// TIA Portal V17 export
// export: Created 2024-09-02T12:50:15.0745708Z, ExportSetting WithDefaults, DisplayName Totally Integrated Automation Portal, DisplayVersion V17, DisplayName TIA Portal Openness, DisplayVersion V17, DisplayName TIA Portal Version Control Interface, DisplayVersion V17, DisplayName STEP 7 Professional, DisplayVersion V17, DisplayName STEP 7 Safety, DisplayVersion V17, DisplayName WinCC Professional, DisplayVersion V17
FUNCTION "AnwFC_ZP_OperatingModes_OP70" : Void   // FC61, LAD
TITLE = FC Operating modes / FC Betriebsarten
{ S7_Optimized_Access := 'TRUE' }
AUTHOR : OlegFuehrus
FAMILY : BA
NAME : BA
VERSION : 0.0
// stored: AutoNumber true, IsIECCheckEnabled false, SetENOAutomatically false, UDAEnableTagReadback false
   VAR_TEMP
      t_e_stop_ok : Bool;
      Dummy : Bool;
   END_VAR
   VAR_TEMP   // added for the SCL form of the ladder/FBD networks
      _w1 : Bool;
      _w2 : Bool;
      _w3 : Bool;
      _w4 : Bool;
      _w5 : Bool;
      _w6 : Bool;
   END_VAR
BEGIN

REGION Network 1: Station lighting On / Stationbeleuchtung Ein
END_REGION

REGION Network 2: Maschine Off (+S-KFK0) / Maschine Aus (+S-KFK0)
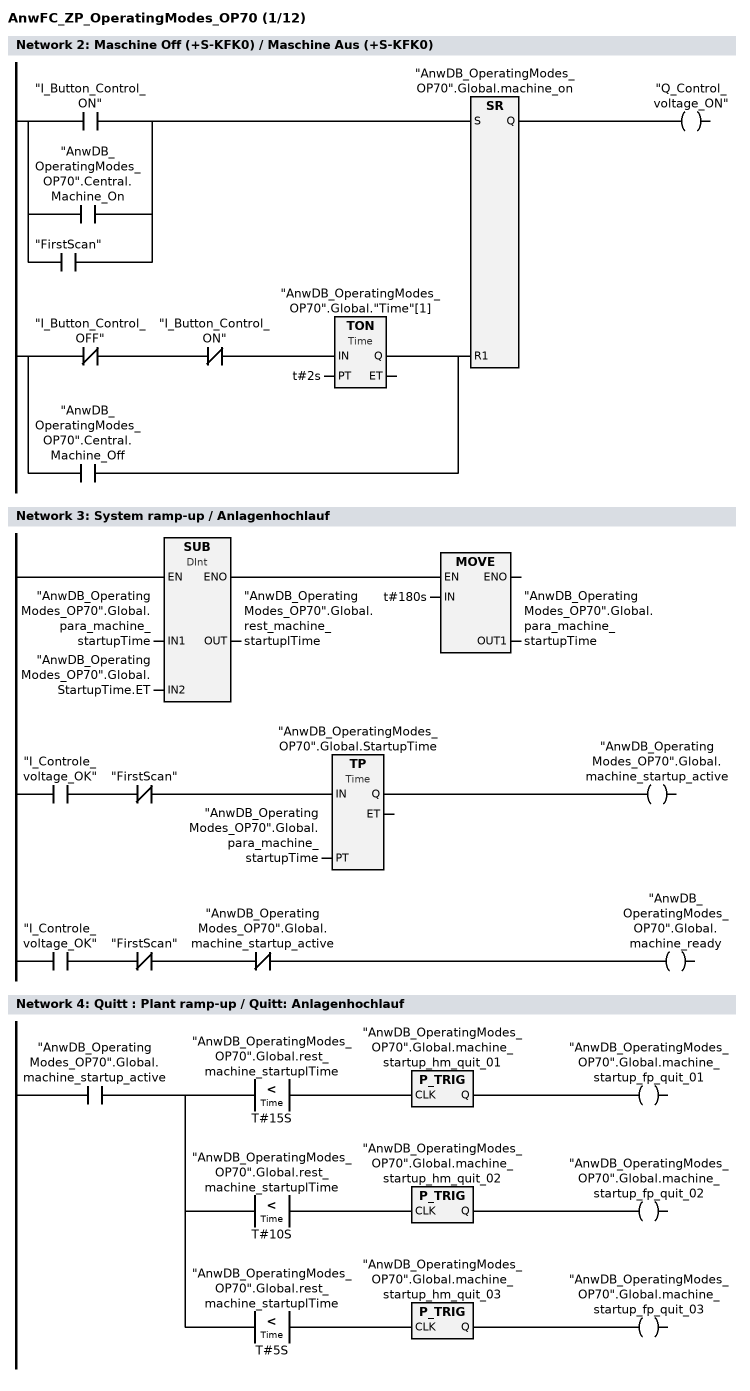
   RUNG wire#powerrail
      Contact( "I_Button_Control_ON" )
      wire#w1
      S_SR(operand := "AnwDB_OperatingModes_OP70".Global.machine_on, r1 := wire#w2)
      Coil( "Q_Control_voltage_ON" )
   END_RUNG
   RUNG wire#powerrail
      Contact( "AnwDB_OperatingModes_OP70".Central.Machine_On )
   END_RUNG wire#w1
   RUNG wire#powerrail
      Contact( "FirstScan" )
   END_RUNG wire#w1
   RUNG wire#powerrail
      I_Contact( "I_Button_Control_OFF" )
      I_Contact( "I_Button_Control_ON" )
      { S7_Templates := "time_type := Time" } "AnwDB_OperatingModes_OP70".Global."Time"[1].TON(pt := t#2s, et =>)
   END_RUNG wire#w2
   RUNG wire#powerrail
      Contact( "AnwDB_OperatingModes_OP70".Central.Machine_Off )
   END_RUNG wire#w2
   // the same network as SCL:
   "AnwDB_OperatingModes_OP70".Global."Time"[1].TON(IN := NOT "I_Button_Control_OFF" AND NOT "I_Button_Control_ON",
                           PT := t#2s);
   IF "I_Button_Control_ON" OR "AnwDB_OperatingModes_OP70".Central.Machine_On OR "FirstScan" THEN
       "AnwDB_OperatingModes_OP70".Global.machine_on := TRUE;   // SR flip-flop
   END_IF;
   IF "AnwDB_OperatingModes_OP70".Global."Time"[1].Q OR "AnwDB_OperatingModes_OP70".Central.Machine_Off THEN
       "AnwDB_OperatingModes_OP70".Global.machine_on := FALSE;
   END_IF;
   "Q_Control_voltage_ON" := "AnwDB_OperatingModes_OP70".Global.machine_on;
END_REGION

REGION Network 3: System ramp-up / Anlagenhochlauf
   RUNG wire#powerrail
      { S7_Templates := "SrcType := DInt" } Sub(in1 := "AnwDB_OperatingModes_OP70".Global.para_machine_startupTime, in2 := "AnwDB_OperatingModes_OP70".Global.StartupTime.ET, out => "AnwDB_OperatingModes_OP70".Global.rest_machine_startuplTime)
      Move(in := t#180s, out1 => "AnwDB_OperatingModes_OP70".Global.para_machine_startupTime)
   END_RUNG
   RUNG wire#powerrail
      Contact( "I_Controle_voltage_OK" )
      I_Contact( "FirstScan" )
      { S7_Templates := "time_type := Time" } "AnwDB_OperatingModes_OP70".Global.StartupTime.TP(pt := "AnwDB_OperatingModes_OP70".Global.para_machine_startupTime, et =>)
      Coil( "AnwDB_OperatingModes_OP70".Global.machine_startup_active )
   END_RUNG
   RUNG wire#powerrail
      Contact( "I_Controle_voltage_OK" )
      I_Contact( "FirstScan" )
      I_Contact( "AnwDB_OperatingModes_OP70".Global.machine_startup_active )
      Coil( "AnwDB_OperatingModes_OP70".Global.machine_ready )
   END_RUNG
   // the same network as SCL:
   "AnwDB_OperatingModes_OP70".Global.rest_machine_startuplTime := "AnwDB_OperatingModes_OP70".Global.para_machine_startupTime - "AnwDB_OperatingModes_OP70".Global.StartupTime.ET;
   "AnwDB_OperatingModes_OP70".Global.para_machine_startupTime := t#180s;
   "AnwDB_OperatingModes_OP70".Global.StartupTime.TP(IN := "I_Controle_voltage_OK" AND NOT "FirstScan",
                           PT := "AnwDB_OperatingModes_OP70".Global.para_machine_startupTime);
   "AnwDB_OperatingModes_OP70".Global.machine_startup_active := "AnwDB_OperatingModes_OP70".Global.StartupTime.Q;
   "AnwDB_OperatingModes_OP70".Global.machine_ready := "I_Controle_voltage_OK" AND NOT "FirstScan" AND NOT "AnwDB_OperatingModes_OP70".Global.machine_startup_active;
END_REGION

REGION Network 4: Quitt : Plant ramp-up / Quitt: Anlagenhochlauf
   RUNG wire#powerrail
      Contact( "AnwDB_OperatingModes_OP70".Global.machine_startup_active )
      wire#w1
      { S7_Templates := "SrcType := Time" } LT_Contact(in1 := "AnwDB_OperatingModes_OP70".Global.rest_machine_startuplTime, in2 := T#15S)
      P_Trig( "AnwDB_OperatingModes_OP70".Global.machine_startup_hm_quit_01 )
      Coil( "AnwDB_OperatingModes_OP70".Global.machine_startup_fp_quit_01 )
   END_RUNG
   RUNG wire#w1
      { S7_Templates := "SrcType := Time" } LT_Contact(in1 := "AnwDB_OperatingModes_OP70".Global.rest_machine_startuplTime, in2 := T#10S)
      P_Trig( "AnwDB_OperatingModes_OP70".Global.machine_startup_hm_quit_02 )
      Coil( "AnwDB_OperatingModes_OP70".Global.machine_startup_fp_quit_02 )
   END_RUNG
   RUNG wire#w1
      { S7_Templates := "SrcType := Time" } LT_Contact(in1 := "AnwDB_OperatingModes_OP70".Global.rest_machine_startuplTime, in2 := T#5S)
      P_Trig( "AnwDB_OperatingModes_OP70".Global.machine_startup_hm_quit_03 )
      Coil( "AnwDB_OperatingModes_OP70".Global.machine_startup_fp_quit_03 )
   END_RUNG
   // the same network as SCL:
   #_w1 := "AnwDB_OperatingModes_OP70".Global.machine_startup_active AND ("AnwDB_OperatingModes_OP70".Global.rest_machine_startuplTime < T#15S);
   #_w2 := #_w1 AND NOT "AnwDB_OperatingModes_OP70".Global.machine_startup_hm_quit_01;   // rising edge
   "AnwDB_OperatingModes_OP70".Global.machine_startup_hm_quit_01 := #_w1;
   "AnwDB_OperatingModes_OP70".Global.machine_startup_fp_quit_01 := #_w2;
   #_w3 := "AnwDB_OperatingModes_OP70".Global.machine_startup_active AND ("AnwDB_OperatingModes_OP70".Global.rest_machine_startuplTime < T#10S);
   #_w4 := #_w3 AND NOT "AnwDB_OperatingModes_OP70".Global.machine_startup_hm_quit_02;   // rising edge
   "AnwDB_OperatingModes_OP70".Global.machine_startup_hm_quit_02 := #_w3;
   "AnwDB_OperatingModes_OP70".Global.machine_startup_fp_quit_02 := #_w4;
   #_w5 := "AnwDB_OperatingModes_OP70".Global.machine_startup_active AND ("AnwDB_OperatingModes_OP70".Global.rest_machine_startuplTime < T#5S);
   #_w6 := #_w5 AND NOT "AnwDB_OperatingModes_OP70".Global.machine_startup_hm_quit_03;   // rising edge
   "AnwDB_OperatingModes_OP70".Global.machine_startup_hm_quit_03 := #_w5;
   "AnwDB_OperatingModes_OP70".Global.machine_startup_fp_quit_03 := #_w6;
END_REGION

REGION Network 5: Starting conditions Ready / Startvoraussetzungen Bereit
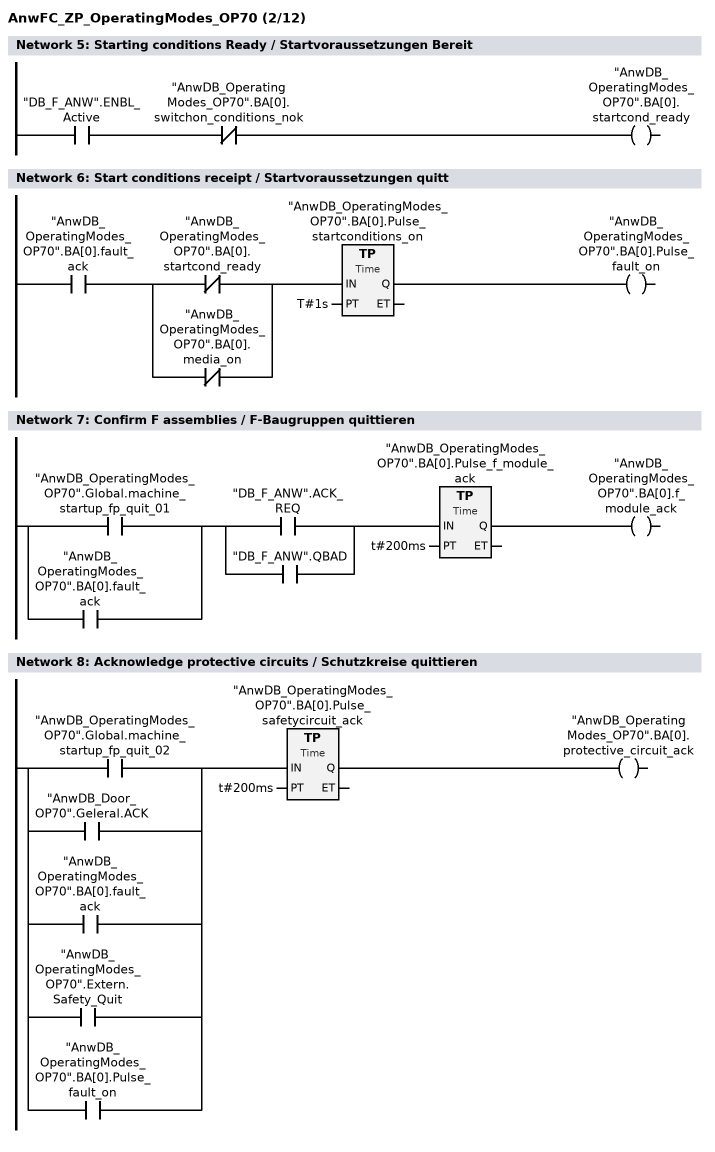
   RUNG wire#powerrail
      Contact( "DB_F_ANW".ENBL_Active )
      I_Contact( "AnwDB_OperatingModes_OP70".BA[0].switchon_conditions_nok )
      Coil( "AnwDB_OperatingModes_OP70".BA[0].startcond_ready )
   END_RUNG
   // the same network as SCL:
   "AnwDB_OperatingModes_OP70".BA[0].startcond_ready := "DB_F_ANW".ENBL_Active AND NOT "AnwDB_OperatingModes_OP70".BA[0].switchon_conditions_nok;
END_REGION

REGION Network 6: Start conditions receipt / Startvoraussetzungen quitt
   RUNG wire#powerrail
      Contact( "AnwDB_OperatingModes_OP70".BA[0].fault_ack )
      wire#w1
      I_Contact( "AnwDB_OperatingModes_OP70".BA[0].startcond_ready )
      wire#w2
      { S7_Templates := "time_type := Time" } "AnwDB_OperatingModes_OP70".BA[0].Pulse_startconditions_on.TP(pt := T#1s, et =>)
      Coil( "AnwDB_OperatingModes_OP70".BA[0].Pulse_fault_on )
   END_RUNG
   RUNG wire#w1
      I_Contact( "AnwDB_OperatingModes_OP70".BA[0].media_on )
   END_RUNG wire#w2
   // the same network as SCL:
   "AnwDB_OperatingModes_OP70".BA[0].Pulse_startconditions_on.TP(IN := "AnwDB_OperatingModes_OP70".BA[0].fault_ack AND (NOT "AnwDB_OperatingModes_OP70".BA[0].startcond_ready OR NOT "AnwDB_OperatingModes_OP70".BA[0].media_on),
                           PT := T#1s);
   "AnwDB_OperatingModes_OP70".BA[0].Pulse_fault_on := "AnwDB_OperatingModes_OP70".BA[0].Pulse_startconditions_on.Q;
END_REGION

REGION Network 7: Confirm F assemblies / F-Baugruppen quittieren
   RUNG wire#powerrail
      Contact( "AnwDB_OperatingModes_OP70".Global.machine_startup_fp_quit_01 )
      wire#w1
      Contact( "DB_F_ANW".ACK_REQ )
      wire#w2
      { S7_Templates := "time_type := Time" } "AnwDB_OperatingModes_OP70".BA[0].Pulse_f_module_ack.TP(pt := t#200ms, et =>)
      Coil( "AnwDB_OperatingModes_OP70".BA[0].f_module_ack )
   END_RUNG
   RUNG wire#powerrail
      Contact( "AnwDB_OperatingModes_OP70".BA[0].fault_ack )
   END_RUNG wire#w1
   RUNG wire#w1
      Contact( "DB_F_ANW".QBAD )
   END_RUNG wire#w2
   // the same network as SCL:
   "AnwDB_OperatingModes_OP70".BA[0].Pulse_f_module_ack.TP(IN := ("AnwDB_OperatingModes_OP70".Global.machine_startup_fp_quit_01 OR "AnwDB_OperatingModes_OP70".BA[0].fault_ack) AND ("DB_F_ANW".ACK_REQ OR "DB_F_ANW".QBAD),
                           PT := t#200ms);
   "AnwDB_OperatingModes_OP70".BA[0].f_module_ack := "AnwDB_OperatingModes_OP70".BA[0].Pulse_f_module_ack.Q;
END_REGION

REGION Network 8: Acknowledge protective circuits / Schutzkreise quittieren
   RUNG wire#powerrail
      Contact( "AnwDB_OperatingModes_OP70".Global.machine_startup_fp_quit_02 )
      wire#w1
      { S7_Templates := "time_type := Time" } "AnwDB_OperatingModes_OP70".BA[0].Pulse_safetycircuit_ack.TP(pt := t#200ms, et =>)
      Coil( "AnwDB_OperatingModes_OP70".BA[0].protective_circuit_ack )
   END_RUNG
   RUNG wire#powerrail
      Contact( "AnwDB_Door_OP70".Geleral.ACK )
   END_RUNG wire#w1
   RUNG wire#powerrail
      Contact( "AnwDB_OperatingModes_OP70".BA[0].fault_ack )
   END_RUNG wire#w1
   RUNG wire#powerrail
      Contact( "AnwDB_OperatingModes_OP70".Extern.Safety_Quit )
   END_RUNG wire#w1
   RUNG wire#powerrail
      Contact( "AnwDB_OperatingModes_OP70".BA[0].Pulse_fault_on )
   END_RUNG wire#w1
   // the same network as SCL:
   "AnwDB_OperatingModes_OP70".BA[0].Pulse_safetycircuit_ack.TP(IN := "AnwDB_OperatingModes_OP70".Global.machine_startup_fp_quit_02 OR "AnwDB_Door_OP70".Geleral.ACK OR "AnwDB_OperatingModes_OP70".BA[0].fault_ack OR "AnwDB_OperatingModes_OP70".Extern.Safety_Quit OR "AnwDB_OperatingModes_OP70".BA[0].Pulse_fault_on,
                           PT := t#200ms);
   "AnwDB_OperatingModes_OP70".BA[0].protective_circuit_ack := "AnwDB_OperatingModes_OP70".BA[0].Pulse_safetycircuit_ack.Q;
END_REGION

REGION Network 9: Fault Acknowledge / Störung quitt
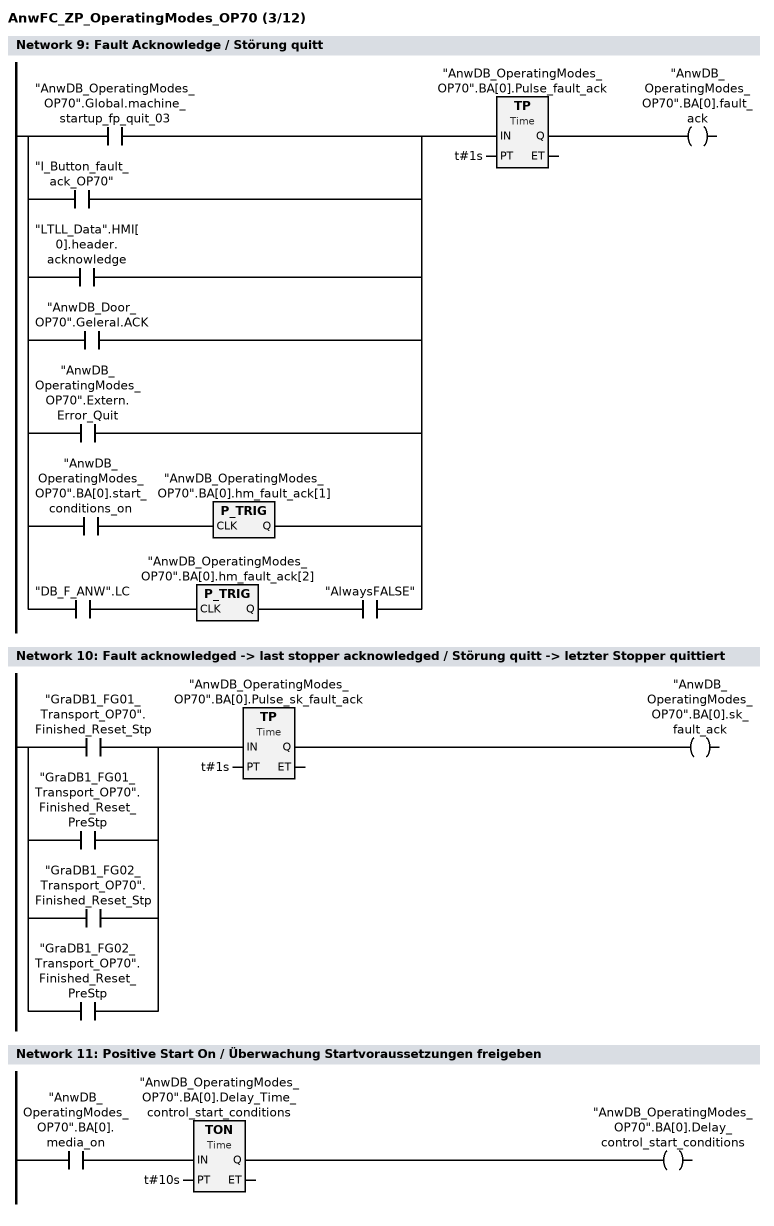
   RUNG wire#powerrail
      Contact( "AnwDB_OperatingModes_OP70".Global.machine_startup_fp_quit_03 )
      wire#w1
      { S7_Templates := "time_type := Time" } "AnwDB_OperatingModes_OP70".BA[0].Pulse_fault_ack.TP(pt := t#1s, et =>)
      Coil( "AnwDB_OperatingModes_OP70".BA[0].fault_ack )
   END_RUNG
   RUNG wire#powerrail
      Contact( "I_Button_fault_ack_OP70" )
   END_RUNG wire#w1
   RUNG wire#powerrail
      Contact( "LTLL_Data".HMI[0].header.acknowledge )
   END_RUNG wire#w1
   RUNG wire#powerrail
      Contact( "AnwDB_Door_OP70".Geleral.ACK )
   END_RUNG wire#w1
   RUNG wire#powerrail
      Contact( "AnwDB_OperatingModes_OP70".Extern.Error_Quit )
   END_RUNG wire#w1
   RUNG wire#powerrail
      Contact( "AnwDB_OperatingModes_OP70".BA[0].start_conditions_on )
      P_Trig( "AnwDB_OperatingModes_OP70".BA[0].hm_fault_ack[1] )
   END_RUNG wire#w1
   RUNG wire#powerrail
      Contact( "DB_F_ANW".LC )
      P_Trig( "AnwDB_OperatingModes_OP70".BA[0].hm_fault_ack[2] )
      Contact( "AlwaysFALSE" )
   END_RUNG wire#w1
   // the same network as SCL:
   #_w1 := "AnwDB_OperatingModes_OP70".BA[0].start_conditions_on;
   #_w2 := #_w1 AND NOT "AnwDB_OperatingModes_OP70".BA[0].hm_fault_ack[1];   // rising edge
   "AnwDB_OperatingModes_OP70".BA[0].hm_fault_ack[1] := #_w1;
   #_w3 := "DB_F_ANW".LC AND NOT "AnwDB_OperatingModes_OP70".BA[0].hm_fault_ack[2];   // rising edge
   "AnwDB_OperatingModes_OP70".BA[0].hm_fault_ack[2] := "DB_F_ANW".LC;
   "AnwDB_OperatingModes_OP70".BA[0].Pulse_fault_ack.TP(IN := "AnwDB_OperatingModes_OP70".Global.machine_startup_fp_quit_03 OR "I_Button_fault_ack_OP70" OR "LTLL_Data".HMI[0].header.acknowledge OR "AnwDB_Door_OP70".Geleral.ACK OR "AnwDB_OperatingModes_OP70".Extern.Error_Quit OR #_w2 OR (#_w3 AND "AlwaysFALSE"),
                           PT := t#1s);
   "AnwDB_OperatingModes_OP70".BA[0].fault_ack := "AnwDB_OperatingModes_OP70".BA[0].Pulse_fault_ack.Q;
END_REGION

REGION Network 10: Fault acknowledged -> last stopper acknowledged / Störung quitt -> letzter Stopper quittiert
   RUNG wire#powerrail
      Contact( "GraDB1_FG01_Transport_OP70".Finished_Reset_Stp )
      wire#w1
      { S7_Templates := "time_type := Time" } "AnwDB_OperatingModes_OP70".BA[0].Pulse_sk_fault_ack.TP(pt := t#1s, et =>)
      Coil( "AnwDB_OperatingModes_OP70".BA[0].sk_fault_ack )
   END_RUNG
   RUNG wire#powerrail
      Contact( "GraDB1_FG01_Transport_OP70".Finished_Reset_PreStp )
   END_RUNG wire#w1
   RUNG wire#powerrail
      Contact( "GraDB1_FG02_Transport_OP70".Finished_Reset_Stp )
   END_RUNG wire#w1
   RUNG wire#powerrail
      Contact( "GraDB1_FG02_Transport_OP70".Finished_Reset_PreStp )
   END_RUNG wire#w1
   // the same network as SCL:
   "AnwDB_OperatingModes_OP70".BA[0].Pulse_sk_fault_ack.TP(IN := "GraDB1_FG01_Transport_OP70".Finished_Reset_Stp OR "GraDB1_FG01_Transport_OP70".Finished_Reset_PreStp OR "GraDB1_FG02_Transport_OP70".Finished_Reset_Stp OR "GraDB1_FG02_Transport_OP70".Finished_Reset_PreStp,
                           PT := t#1s);
   "AnwDB_OperatingModes_OP70".BA[0].sk_fault_ack := "AnwDB_OperatingModes_OP70".BA[0].Pulse_sk_fault_ack.Q;
END_REGION

REGION Network 11: Positive Start On / Überwachung Startvoraussetzungen freigeben
   RUNG wire#powerrail
      Contact( "AnwDB_OperatingModes_OP70".BA[0].media_on )
      { S7_Templates := "time_type := Time" } "AnwDB_OperatingModes_OP70".BA[0].Delay_Time_control_start_conditions.TON(pt := t#10s, et =>)
      Coil( "AnwDB_OperatingModes_OP70".BA[0].Delay_control_start_conditions )
   END_RUNG
   // the same network as SCL:
   "AnwDB_OperatingModes_OP70".BA[0].Delay_Time_control_start_conditions.TON(IN := "AnwDB_OperatingModes_OP70".BA[0].media_on,
                           PT := t#10s);
   "AnwDB_OperatingModes_OP70".BA[0].Delay_control_start_conditions := "AnwDB_OperatingModes_OP70".BA[0].Delay_Time_control_start_conditions.Q;
END_REGION

REGION Network 12: Starting conditions are ON / Startvoraussetzungen sind ein
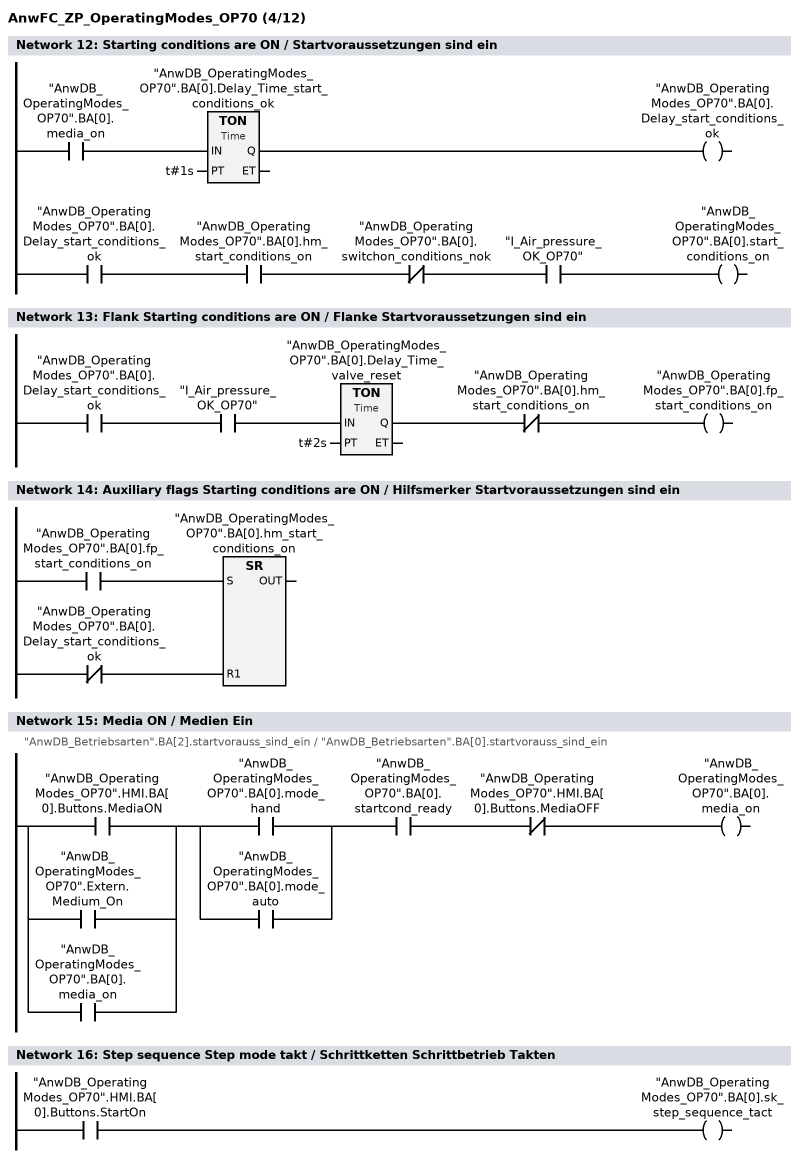
   RUNG wire#powerrail
      Contact( "AnwDB_OperatingModes_OP70".BA[0].media_on )
      { S7_Templates := "time_type := Time" } "AnwDB_OperatingModes_OP70".BA[0].Delay_Time_start_conditions_ok.TON(pt := t#1s, et =>)
      Coil( "AnwDB_OperatingModes_OP70".BA[0].Delay_start_conditions_ok )
   END_RUNG
   RUNG wire#powerrail
      Contact( "AnwDB_OperatingModes_OP70".BA[0].Delay_start_conditions_ok )
      Contact( "AnwDB_OperatingModes_OP70".BA[0].hm_start_conditions_on )
      I_Contact( "AnwDB_OperatingModes_OP70".BA[0].switchon_conditions_nok )
      Contact( "I_Air_pressure_OK_OP70" )
      Coil( "AnwDB_OperatingModes_OP70".BA[0].start_conditions_on )
   END_RUNG
   // the same network as SCL:
   "AnwDB_OperatingModes_OP70".BA[0].Delay_Time_start_conditions_ok.TON(IN := "AnwDB_OperatingModes_OP70".BA[0].media_on,
                           PT := t#1s);
   "AnwDB_OperatingModes_OP70".BA[0].Delay_start_conditions_ok := "AnwDB_OperatingModes_OP70".BA[0].Delay_Time_start_conditions_ok.Q;
   "AnwDB_OperatingModes_OP70".BA[0].start_conditions_on := "AnwDB_OperatingModes_OP70".BA[0].Delay_start_conditions_ok AND "AnwDB_OperatingModes_OP70".BA[0].hm_start_conditions_on AND NOT "AnwDB_OperatingModes_OP70".BA[0].switchon_conditions_nok AND "I_Air_pressure_OK_OP70";
END_REGION

REGION Network 13: Flank Starting conditions are ON / Flanke Startvoraussetzungen sind ein
   RUNG wire#powerrail
      Contact( "AnwDB_OperatingModes_OP70".BA[0].Delay_start_conditions_ok )
      Contact( "I_Air_pressure_OK_OP70" )
      { S7_Templates := "time_type := Time" } "AnwDB_OperatingModes_OP70".BA[0].Delay_Time_valve_reset.TON(pt := t#2s, et =>)
      I_Contact( "AnwDB_OperatingModes_OP70".BA[0].hm_start_conditions_on )
      Coil( "AnwDB_OperatingModes_OP70".BA[0].fp_start_conditions_on )
   END_RUNG
   // the same network as SCL:
   "AnwDB_OperatingModes_OP70".BA[0].Delay_Time_valve_reset.TON(IN := "AnwDB_OperatingModes_OP70".BA[0].Delay_start_conditions_ok AND "I_Air_pressure_OK_OP70",
                           PT := t#2s);
   "AnwDB_OperatingModes_OP70".BA[0].fp_start_conditions_on := "AnwDB_OperatingModes_OP70".BA[0].Delay_Time_valve_reset.Q AND NOT "AnwDB_OperatingModes_OP70".BA[0].hm_start_conditions_on;
END_REGION

REGION Network 14: Auxiliary flags Starting conditions are ON / Hilfsmerker Startvoraussetzungen sind ein
   RUNG wire#powerrail
      Contact( "AnwDB_OperatingModes_OP70".BA[0].fp_start_conditions_on )
      S_SR(operand := "AnwDB_OperatingModes_OP70".BA[0].hm_start_conditions_on, r1 := wire#w1)
   END_RUNG
   RUNG wire#powerrail
      I_Contact( "AnwDB_OperatingModes_OP70".BA[0].Delay_start_conditions_ok )
   END_RUNG wire#w1
   // the same network as SCL:
   #_w1 := NOT "AnwDB_OperatingModes_OP70".BA[0].Delay_start_conditions_ok;
   IF "AnwDB_OperatingModes_OP70".BA[0].fp_start_conditions_on THEN
       "AnwDB_OperatingModes_OP70".BA[0].hm_start_conditions_on := TRUE;   // SR flip-flop
   END_IF;
   IF #_w1 THEN "AnwDB_OperatingModes_OP70".BA[0].hm_start_conditions_on := FALSE; END_IF;
END_REGION

REGION Network 15: Media ON / Medien Ein
   // "AnwDB_Betriebsarten".BA[2].startvorauss_sind_ein / "AnwDB_Betriebsarten".BA[0].startvorauss_sind_ein
   RUNG wire#powerrail
      Contact( "AnwDB_OperatingModes_OP70".HMI.BA[0].Buttons.MediaON )
      wire#w1
      Contact( "AnwDB_OperatingModes_OP70".BA[0].mode_hand )
      wire#w2
      Contact( "AnwDB_OperatingModes_OP70".BA[0].startcond_ready )
      I_Contact( "AnwDB_OperatingModes_OP70".HMI.BA[0].Buttons.MediaOFF )
      Coil( "AnwDB_OperatingModes_OP70".BA[0].media_on )
   END_RUNG
   RUNG wire#powerrail
      Contact( "AnwDB_OperatingModes_OP70".Extern.Medium_On )
   END_RUNG wire#w1
   RUNG wire#powerrail
      Contact( "AnwDB_OperatingModes_OP70".BA[0].media_on )
   END_RUNG wire#w1
   RUNG wire#w1
      Contact( "AnwDB_OperatingModes_OP70".BA[0].mode_auto )
   END_RUNG wire#w2
   // the same network as SCL:
   "AnwDB_OperatingModes_OP70".BA[0].media_on := ("AnwDB_OperatingModes_OP70".HMI.BA[0].Buttons.MediaON OR "AnwDB_OperatingModes_OP70".Extern.Medium_On OR "AnwDB_OperatingModes_OP70".BA[0].media_on) AND ("AnwDB_OperatingModes_OP70".BA[0].mode_hand OR "AnwDB_OperatingModes_OP70".BA[0].mode_auto) AND "AnwDB_OperatingModes_OP70".BA[0].startcond_ready AND NOT "AnwDB_OperatingModes_OP70".HMI.BA[0].Buttons.MediaOFF;
END_REGION

REGION Network 16: Step sequence Step mode takt / Schrittketten Schrittbetrieb Takten
   RUNG wire#powerrail
      Contact( "AnwDB_OperatingModes_OP70".HMI.BA[0].Buttons.StartOn )
      Coil( "AnwDB_OperatingModes_OP70".BA[0].sk_step_sequence_tact )
   END_RUNG
   // the same network as SCL:
   "AnwDB_OperatingModes_OP70".BA[0].sk_step_sequence_tact := "AnwDB_OperatingModes_OP70".HMI.BA[0].Buttons.StartOn;
END_REGION

REGION Network 17: Preselection Auto / Vorwahl Automatik
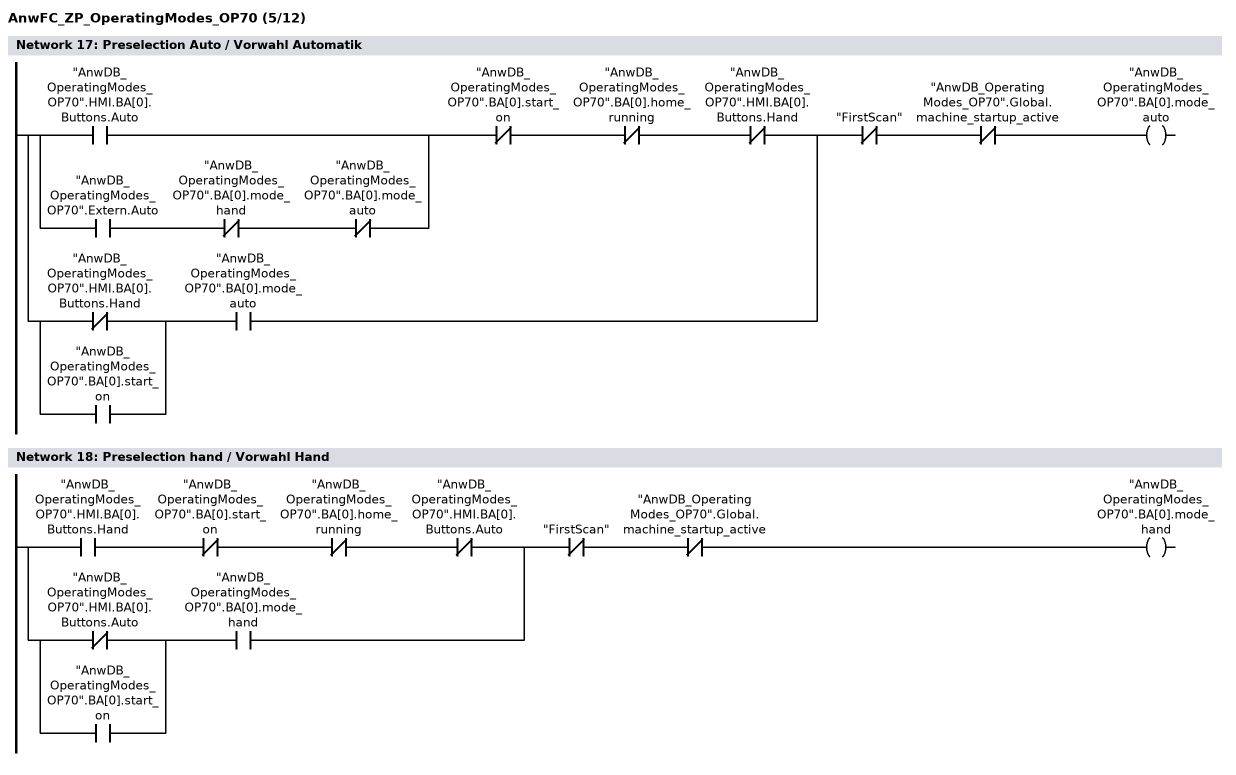
   RUNG wire#powerrail
      Contact( "AnwDB_OperatingModes_OP70".HMI.BA[0].Buttons.Auto )
      wire#w1
      I_Contact( "AnwDB_OperatingModes_OP70".BA[0].start_on )
      I_Contact( "AnwDB_OperatingModes_OP70".BA[0].home_running )
      I_Contact( "AnwDB_OperatingModes_OP70".HMI.BA[0].Buttons.Hand )
      wire#w2
      I_Contact( "FirstScan" )
      I_Contact( "AnwDB_OperatingModes_OP70".Global.machine_startup_active )
      Coil( "AnwDB_OperatingModes_OP70".BA[0].mode_auto )
   END_RUNG
   RUNG wire#powerrail
      Contact( "AnwDB_OperatingModes_OP70".Extern.Auto )
      I_Contact( "AnwDB_OperatingModes_OP70".BA[0].mode_hand )
      I_Contact( "AnwDB_OperatingModes_OP70".BA[0].mode_auto )
   END_RUNG wire#w1
   RUNG wire#powerrail
      I_Contact( "AnwDB_OperatingModes_OP70".HMI.BA[0].Buttons.Hand )
      wire#w3
      Contact( "AnwDB_OperatingModes_OP70".BA[0].mode_auto )
   END_RUNG wire#w2
   RUNG wire#powerrail
      Contact( "AnwDB_OperatingModes_OP70".BA[0].start_on )
   END_RUNG wire#w3
   // the same network as SCL:
   "AnwDB_OperatingModes_OP70".BA[0].mode_auto := ((("AnwDB_OperatingModes_OP70".HMI.BA[0].Buttons.Auto OR ("AnwDB_OperatingModes_OP70".Extern.Auto AND NOT "AnwDB_OperatingModes_OP70".BA[0].mode_hand AND NOT "AnwDB_OperatingModes_OP70".BA[0].mode_auto)) AND NOT "AnwDB_OperatingModes_OP70".BA[0].start_on AND NOT "AnwDB_OperatingModes_OP70".BA[0].home_running AND NOT "AnwDB_OperatingModes_OP70".HMI.BA[0].Buttons.Hand) OR ((NOT "AnwDB_OperatingModes_OP70".HMI.BA[0].Buttons.Hand OR "AnwDB_OperatingModes_OP70".BA[0].start_on) AND "AnwDB_OperatingModes_OP70".BA[0].mode_auto)) AND NOT "FirstScan" AND NOT "AnwDB_OperatingModes_OP70".Global.machine_startup_active;
END_REGION

REGION Network 18: Preselection hand / Vorwahl Hand
   RUNG wire#powerrail
      Contact( "AnwDB_OperatingModes_OP70".HMI.BA[0].Buttons.Hand )
      I_Contact( "AnwDB_OperatingModes_OP70".BA[0].start_on )
      I_Contact( "AnwDB_OperatingModes_OP70".BA[0].home_running )
      I_Contact( "AnwDB_OperatingModes_OP70".HMI.BA[0].Buttons.Auto )
      wire#w1
      I_Contact( "FirstScan" )
      I_Contact( "AnwDB_OperatingModes_OP70".Global.machine_startup_active )
      Coil( "AnwDB_OperatingModes_OP70".BA[0].mode_hand )
   END_RUNG
   RUNG wire#powerrail
      I_Contact( "AnwDB_OperatingModes_OP70".HMI.BA[0].Buttons.Auto )
      wire#w2
      Contact( "AnwDB_OperatingModes_OP70".BA[0].mode_hand )
   END_RUNG wire#w1
   RUNG wire#powerrail
      Contact( "AnwDB_OperatingModes_OP70".BA[0].start_on )
   END_RUNG wire#w2
   // the same network as SCL:
   "AnwDB_OperatingModes_OP70".BA[0].mode_hand := (("AnwDB_OperatingModes_OP70".HMI.BA[0].Buttons.Hand AND NOT "AnwDB_OperatingModes_OP70".BA[0].start_on AND NOT "AnwDB_OperatingModes_OP70".BA[0].home_running AND NOT "AnwDB_OperatingModes_OP70".HMI.BA[0].Buttons.Auto) OR ((NOT "AnwDB_OperatingModes_OP70".HMI.BA[0].Buttons.Auto OR "AnwDB_OperatingModes_OP70".BA[0].start_on) AND "AnwDB_OperatingModes_OP70".BA[0].mode_hand)) AND NOT "FirstScan" AND NOT "AnwDB_OperatingModes_OP70".Global.machine_startup_active;
END_REGION

REGION Network 19: Start On / Start Ein
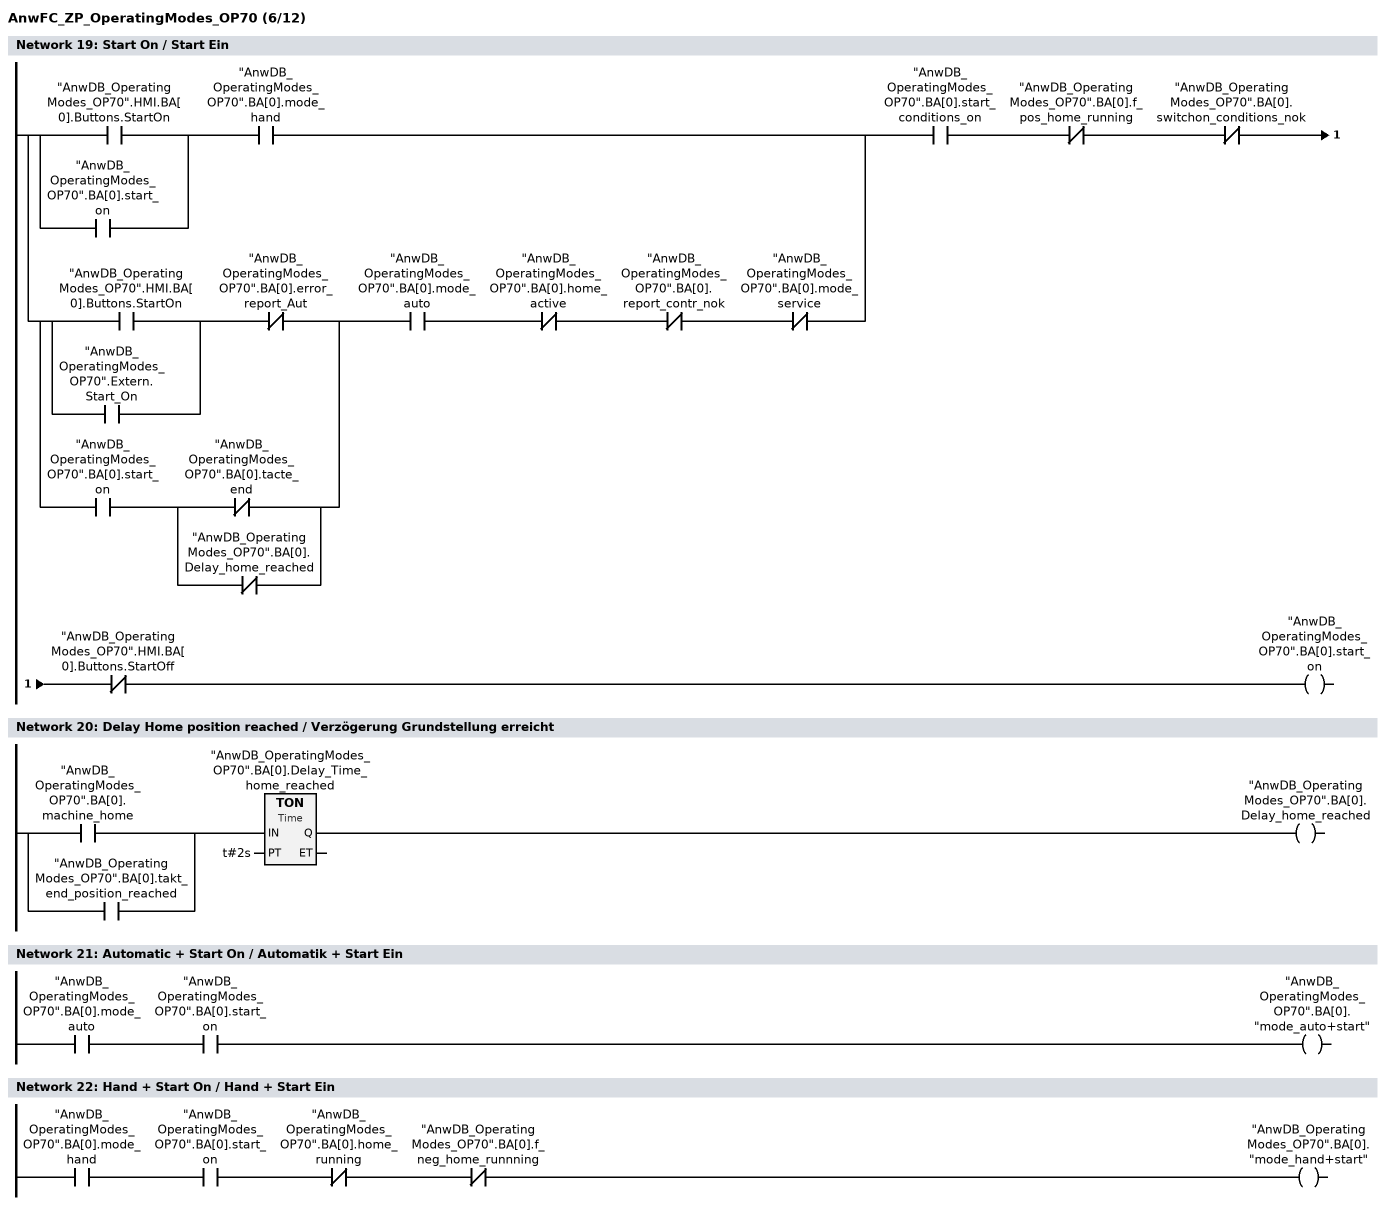
   RUNG wire#powerrail
      Contact( "AnwDB_OperatingModes_OP70".HMI.BA[0].Buttons.StartOn )
      wire#w1
      Contact( "AnwDB_OperatingModes_OP70".BA[0].mode_hand )
      wire#w2
      Contact( "AnwDB_OperatingModes_OP70".BA[0].start_conditions_on )
      I_Contact( "AnwDB_OperatingModes_OP70".BA[0].f_pos_home_running )
      I_Contact( "AnwDB_OperatingModes_OP70".BA[0].switchon_conditions_nok )
      I_Contact( "AnwDB_OperatingModes_OP70".HMI.BA[0].Buttons.StartOff )
      Coil( "AnwDB_OperatingModes_OP70".BA[0].start_on )
   END_RUNG
   RUNG wire#powerrail
      Contact( "AnwDB_OperatingModes_OP70".BA[0].start_on )
   END_RUNG wire#w1
   RUNG wire#powerrail
      Contact( "AnwDB_OperatingModes_OP70".HMI.BA[0].Buttons.StartOn )
      wire#w3
      I_Contact( "AnwDB_OperatingModes_OP70".BA[0].error_report_Aut )
      wire#w4
      Contact( "AnwDB_OperatingModes_OP70".BA[0].mode_auto )
      I_Contact( "AnwDB_OperatingModes_OP70".BA[0].home_active )
      I_Contact( "AnwDB_OperatingModes_OP70".BA[0].report_contr_nok )
      I_Contact( "AnwDB_OperatingModes_OP70".BA[0].mode_service )
   END_RUNG wire#w2
   RUNG wire#powerrail
      Contact( "AnwDB_OperatingModes_OP70".Extern.Start_On )
   END_RUNG wire#w3
   RUNG wire#powerrail
      Contact( "AnwDB_OperatingModes_OP70".BA[0].start_on )
      wire#w5
      I_Contact( "AnwDB_OperatingModes_OP70".BA[0].tacte_end )
   END_RUNG wire#w4
   RUNG wire#w5
      I_Contact( "AnwDB_OperatingModes_OP70".BA[0].Delay_home_reached )
   END_RUNG wire#w4
   // the same network as SCL:
   "AnwDB_OperatingModes_OP70".BA[0].start_on := ((("AnwDB_OperatingModes_OP70".HMI.BA[0].Buttons.StartOn OR "AnwDB_OperatingModes_OP70".BA[0].start_on) AND "AnwDB_OperatingModes_OP70".BA[0].mode_hand) OR (((("AnwDB_OperatingModes_OP70".HMI.BA[0].Buttons.StartOn OR "AnwDB_OperatingModes_OP70".Extern.Start_On) AND NOT "AnwDB_OperatingModes_OP70".BA[0].error_report_Aut) OR ("AnwDB_OperatingModes_OP70".BA[0].start_on AND (NOT "AnwDB_OperatingModes_OP70".BA[0].tacte_end OR NOT "AnwDB_OperatingModes_OP70".BA[0].Delay_home_reached))) AND "AnwDB_OperatingModes_OP70".BA[0].mode_auto AND NOT "AnwDB_OperatingModes_OP70".BA[0].home_active AND NOT "AnwDB_OperatingModes_OP70".BA[0].report_contr_nok AND NOT "AnwDB_OperatingModes_OP70".BA[0].mode_service)) AND "AnwDB_OperatingModes_OP70".BA[0].start_conditions_on AND NOT "AnwDB_OperatingModes_OP70".BA[0].f_pos_home_running AND NOT "AnwDB_OperatingModes_OP70".BA[0].switchon_conditions_nok AND NOT "AnwDB_OperatingModes_OP70".HMI.BA[0].Buttons.StartOff;
END_REGION

REGION Network 20: Delay Home position reached / Verzögerung Grundstellung erreicht
   RUNG wire#powerrail
      Contact( "AnwDB_OperatingModes_OP70".BA[0].machine_home )
      wire#w1
      { S7_Templates := "time_type := Time" } "AnwDB_OperatingModes_OP70".BA[0].Delay_Time_home_reached.TON(pt := t#2s, et =>)
      Coil( "AnwDB_OperatingModes_OP70".BA[0].Delay_home_reached )
   END_RUNG
   RUNG wire#powerrail
      Contact( "AnwDB_OperatingModes_OP70".BA[0].takt_end_position_reached )
   END_RUNG wire#w1
   // the same network as SCL:
   "AnwDB_OperatingModes_OP70".BA[0].Delay_Time_home_reached.TON(IN := "AnwDB_OperatingModes_OP70".BA[0].machine_home OR "AnwDB_OperatingModes_OP70".BA[0].takt_end_position_reached,
                           PT := t#2s);
   "AnwDB_OperatingModes_OP70".BA[0].Delay_home_reached := "AnwDB_OperatingModes_OP70".BA[0].Delay_Time_home_reached.Q;
END_REGION

REGION Network 21: Automatic + Start On / Automatik + Start Ein
   RUNG wire#powerrail
      Contact( "AnwDB_OperatingModes_OP70".BA[0].mode_auto )
      Contact( "AnwDB_OperatingModes_OP70".BA[0].start_on )
      Coil( "AnwDB_OperatingModes_OP70".BA[0]."mode_auto+start" )
   END_RUNG
   // the same network as SCL:
   "AnwDB_OperatingModes_OP70".BA[0]."mode_auto+start" := "AnwDB_OperatingModes_OP70".BA[0].mode_auto AND "AnwDB_OperatingModes_OP70".BA[0].start_on;
END_REGION

REGION Network 22: Hand + Start On / Hand + Start Ein
   RUNG wire#powerrail
      Contact( "AnwDB_OperatingModes_OP70".BA[0].mode_hand )
      Contact( "AnwDB_OperatingModes_OP70".BA[0].start_on )
      I_Contact( "AnwDB_OperatingModes_OP70".BA[0].home_running )
      I_Contact( "AnwDB_OperatingModes_OP70".BA[0].f_neg_home_runnning )
      Coil( "AnwDB_OperatingModes_OP70".BA[0]."mode_hand+start" )
   END_RUNG
   // the same network as SCL:
   "AnwDB_OperatingModes_OP70".BA[0]."mode_hand+start" := "AnwDB_OperatingModes_OP70".BA[0].mode_hand AND "AnwDB_OperatingModes_OP70".BA[0].start_on AND NOT "AnwDB_OperatingModes_OP70".BA[0].home_running AND NOT "AnwDB_OperatingModes_OP70".BA[0].f_neg_home_runnning;
END_REGION

REGION Network 23: Move to home position / Grundstellung anfahren
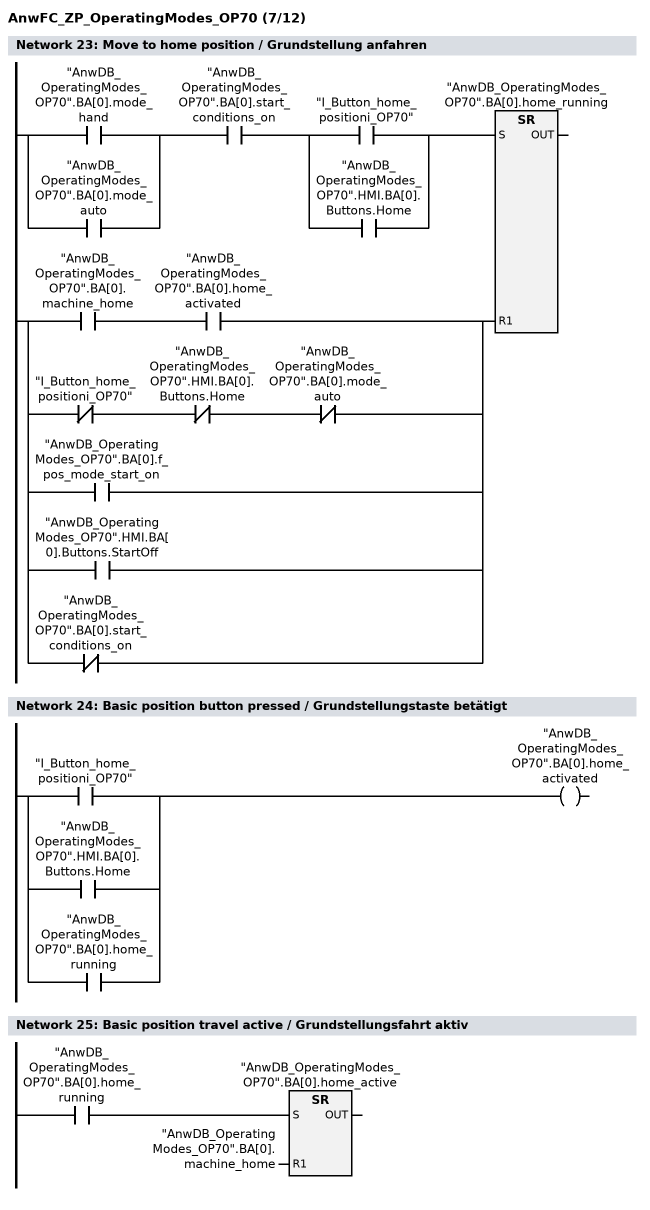
   RUNG wire#powerrail
      Contact( "AnwDB_OperatingModes_OP70".BA[0].mode_hand )
      wire#w1
      Contact( "AnwDB_OperatingModes_OP70".BA[0].start_conditions_on )
      wire#w2
      Contact( "I_Button_home_positioni_OP70" )
      wire#w3
      S_SR(operand := "AnwDB_OperatingModes_OP70".BA[0].home_running, r1 := wire#w4)
   END_RUNG
   RUNG wire#powerrail
      Contact( "AnwDB_OperatingModes_OP70".BA[0].mode_auto )
   END_RUNG wire#w1
   RUNG wire#w2
      Contact( "AnwDB_OperatingModes_OP70".HMI.BA[0].Buttons.Home )
   END_RUNG wire#w3
   RUNG wire#powerrail
      Contact( "AnwDB_OperatingModes_OP70".BA[0].machine_home )
      Contact( "AnwDB_OperatingModes_OP70".BA[0].home_activated )
   END_RUNG wire#w4
   RUNG wire#powerrail
      I_Contact( "I_Button_home_positioni_OP70" )
      I_Contact( "AnwDB_OperatingModes_OP70".HMI.BA[0].Buttons.Home )
      I_Contact( "AnwDB_OperatingModes_OP70".BA[0].mode_auto )
   END_RUNG wire#w4
   RUNG wire#powerrail
      Contact( "AnwDB_OperatingModes_OP70".BA[0].f_pos_mode_start_on )
   END_RUNG wire#w4
   RUNG wire#powerrail
      Contact( "AnwDB_OperatingModes_OP70".HMI.BA[0].Buttons.StartOff )
   END_RUNG wire#w4
   RUNG wire#powerrail
      I_Contact( "AnwDB_OperatingModes_OP70".BA[0].start_conditions_on )
   END_RUNG wire#w4
   // the same network as SCL:
   #_w1 := ("AnwDB_OperatingModes_OP70".BA[0].machine_home AND "AnwDB_OperatingModes_OP70".BA[0].home_activated) OR (NOT "I_Button_home_positioni_OP70" AND NOT "AnwDB_OperatingModes_OP70".HMI.BA[0].Buttons.Home AND NOT "AnwDB_OperatingModes_OP70".BA[0].mode_auto) OR "AnwDB_OperatingModes_OP70".BA[0].f_pos_mode_start_on OR "AnwDB_OperatingModes_OP70".HMI.BA[0].Buttons.StartOff OR NOT "AnwDB_OperatingModes_OP70".BA[0].start_conditions_on;
   IF ("AnwDB_OperatingModes_OP70".BA[0].mode_hand OR "AnwDB_OperatingModes_OP70".BA[0].mode_auto) AND "AnwDB_OperatingModes_OP70".BA[0].start_conditions_on AND ("I_Button_home_positioni_OP70" OR "AnwDB_OperatingModes_OP70".HMI.BA[0].Buttons.Home) THEN
       "AnwDB_OperatingModes_OP70".BA[0].home_running := TRUE;   // SR flip-flop
   END_IF;
   IF #_w1 THEN "AnwDB_OperatingModes_OP70".BA[0].home_running := FALSE; END_IF;
END_REGION

REGION Network 24: Basic position button pressed / Grundstellungstaste betätigt
   RUNG wire#powerrail
      Contact( "I_Button_home_positioni_OP70" )
      wire#w1
      Coil( "AnwDB_OperatingModes_OP70".BA[0].home_activated )
   END_RUNG
   RUNG wire#powerrail
      Contact( "AnwDB_OperatingModes_OP70".HMI.BA[0].Buttons.Home )
   END_RUNG wire#w1
   RUNG wire#powerrail
      Contact( "AnwDB_OperatingModes_OP70".BA[0].home_running )
   END_RUNG wire#w1
   // the same network as SCL:
   "AnwDB_OperatingModes_OP70".BA[0].home_activated := "I_Button_home_positioni_OP70" OR "AnwDB_OperatingModes_OP70".HMI.BA[0].Buttons.Home OR "AnwDB_OperatingModes_OP70".BA[0].home_running;
END_REGION

REGION Network 25: Basic position travel active / Grundstellungsfahrt aktiv
   RUNG wire#powerrail
      Contact( "AnwDB_OperatingModes_OP70".BA[0].home_running )
      S_SR(operand := "AnwDB_OperatingModes_OP70".BA[0].home_active, r1 := "AnwDB_OperatingModes_OP70".BA[0].machine_home)
   END_RUNG
   // the same network as SCL:
   #_w1 := "AnwDB_OperatingModes_OP70".BA[0].machine_home;
   IF "AnwDB_OperatingModes_OP70".BA[0].home_running THEN
       "AnwDB_OperatingModes_OP70".BA[0].home_active := TRUE;   // SR flip-flop
   END_IF;
   IF #_w1 THEN "AnwDB_OperatingModes_OP70".BA[0].home_active := FALSE; END_IF;
END_REGION

REGION Network 26: Preselection stop at the end of tact / Vorwahl Halt bei Taktende
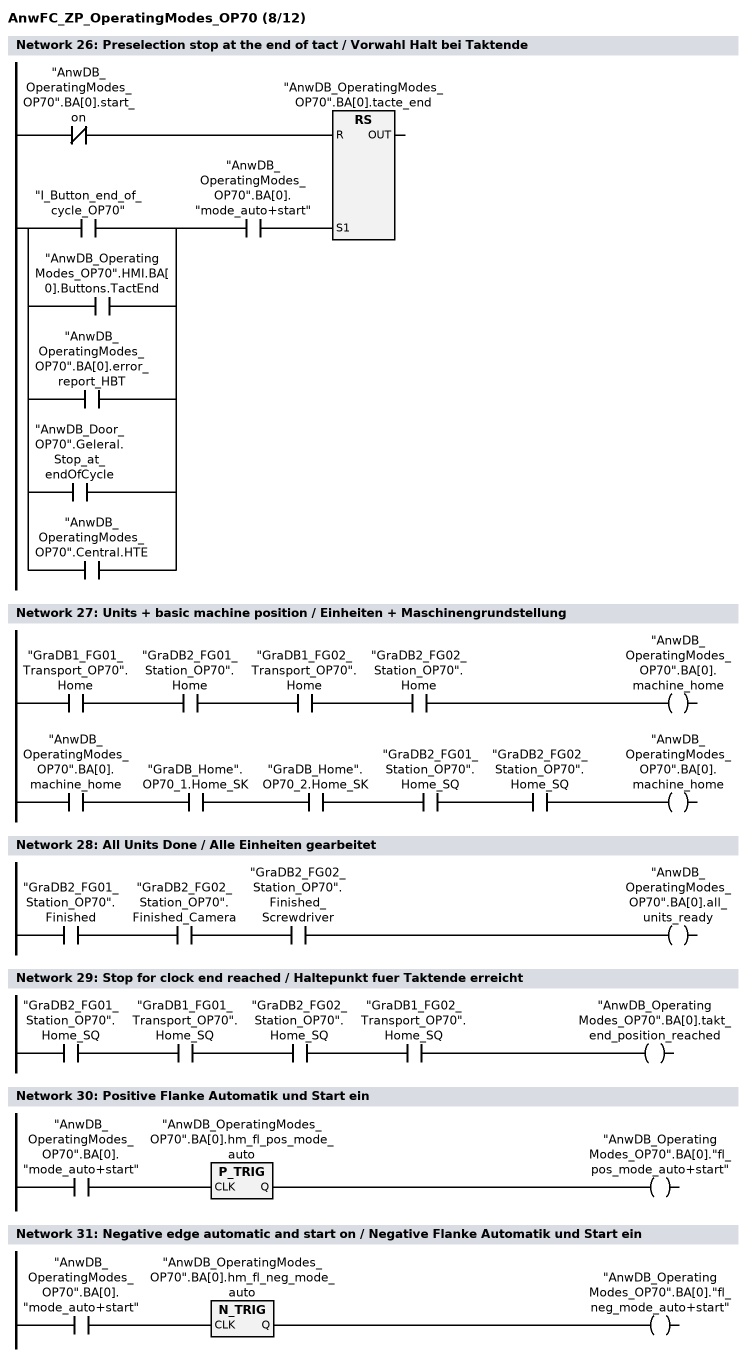
   RUNG wire#powerrail
      I_Contact( "AnwDB_OperatingModes_OP70".BA[0].start_on )
      S_RS(operand := "AnwDB_OperatingModes_OP70".BA[0].tacte_end, s1 := wire#w2)
   END_RUNG
   RUNG wire#powerrail
      Contact( "I_Button_end_of_cycle_OP70" )
      wire#w1
      Contact( "AnwDB_OperatingModes_OP70".BA[0]."mode_auto+start" )
   END_RUNG wire#w2
   RUNG wire#powerrail
      Contact( "AnwDB_OperatingModes_OP70".HMI.BA[0].Buttons.TactEnd )
   END_RUNG wire#w1
   RUNG wire#powerrail
      Contact( "AnwDB_OperatingModes_OP70".BA[0].error_report_HBT )
   END_RUNG wire#w1
   RUNG wire#powerrail
      Contact( "AnwDB_Door_OP70".Geleral.Stop_at_endOfCycle )
   END_RUNG wire#w1
   RUNG wire#powerrail
      Contact( "AnwDB_OperatingModes_OP70".Central.HTE )
   END_RUNG wire#w1
   // the same network as SCL:
   #_w1 := ("I_Button_end_of_cycle_OP70" OR "AnwDB_OperatingModes_OP70".HMI.BA[0].Buttons.TactEnd OR "AnwDB_OperatingModes_OP70".BA[0].error_report_HBT OR "AnwDB_Door_OP70".Geleral.Stop_at_endOfCycle OR "AnwDB_OperatingModes_OP70".Central.HTE) AND "AnwDB_OperatingModes_OP70".BA[0]."mode_auto+start";
   IF NOT "AnwDB_OperatingModes_OP70".BA[0].start_on THEN
       "AnwDB_OperatingModes_OP70".BA[0].tacte_end := FALSE;   // RS flip-flop
   END_IF;
   IF #_w1 THEN "AnwDB_OperatingModes_OP70".BA[0].tacte_end := TRUE; END_IF;
END_REGION

REGION Network 27: Units + basic machine position / Einheiten + Maschinengrundstellung
   RUNG wire#powerrail
      Contact( "GraDB1_FG01_Transport_OP70".Home )
      Contact( "GraDB2_FG01_Station_OP70".Home )
      Contact( "GraDB1_FG02_Transport_OP70".Home )
      Contact( "GraDB2_FG02_Station_OP70".Home )
      Coil( "AnwDB_OperatingModes_OP70".BA[0].machine_home )
   END_RUNG
   RUNG wire#powerrail
      Contact( "AnwDB_OperatingModes_OP70".BA[0].machine_home )
      Contact( "GraDB_Home".OP70_1.Home_SK )
      Contact( "GraDB_Home".OP70_2.Home_SK )
      Contact( "GraDB2_FG01_Station_OP70".Home_SQ )
      Contact( "GraDB2_FG02_Station_OP70".Home_SQ )
      Coil( "AnwDB_OperatingModes_OP70".BA[0].machine_home )
   END_RUNG
   // the same network as SCL:
   "AnwDB_OperatingModes_OP70".BA[0].machine_home := "GraDB1_FG01_Transport_OP70".Home AND "GraDB2_FG01_Station_OP70".Home AND "GraDB1_FG02_Transport_OP70".Home AND "GraDB2_FG02_Station_OP70".Home;
   "AnwDB_OperatingModes_OP70".BA[0].machine_home := "AnwDB_OperatingModes_OP70".BA[0].machine_home AND "GraDB_Home".OP70_1.Home_SK AND "GraDB_Home".OP70_2.Home_SK AND "GraDB2_FG01_Station_OP70".Home_SQ AND "GraDB2_FG02_Station_OP70".Home_SQ;
END_REGION

REGION Network 28: All Units Done / Alle Einheiten gearbeitet
   RUNG wire#powerrail
      Contact( "GraDB2_FG01_Station_OP70".Finished )
      Contact( "GraDB2_FG02_Station_OP70".Finished_Camera )
      Contact( "GraDB2_FG02_Station_OP70".Finished_Screwdriver )
      Coil( "AnwDB_OperatingModes_OP70".BA[0].all_units_ready )
   END_RUNG
   // the same network as SCL:
   "AnwDB_OperatingModes_OP70".BA[0].all_units_ready := "GraDB2_FG01_Station_OP70".Finished AND "GraDB2_FG02_Station_OP70".Finished_Camera AND "GraDB2_FG02_Station_OP70".Finished_Screwdriver;
END_REGION

REGION Network 29: Stop for clock end reached / Haltepunkt fuer Taktende erreicht
   RUNG wire#powerrail
      Contact( "GraDB2_FG01_Station_OP70".Home_SQ )
      Contact( "GraDB1_FG01_Transport_OP70".Home_SQ )
      Contact( "GraDB2_FG02_Station_OP70".Home_SQ )
      Contact( "GraDB1_FG02_Transport_OP70".Home_SQ )
      Coil( "AnwDB_OperatingModes_OP70".BA[0].takt_end_position_reached )
   END_RUNG
   // the same network as SCL:
   "AnwDB_OperatingModes_OP70".BA[0].takt_end_position_reached := "GraDB2_FG01_Station_OP70".Home_SQ AND "GraDB1_FG01_Transport_OP70".Home_SQ AND "GraDB2_FG02_Station_OP70".Home_SQ AND "GraDB1_FG02_Transport_OP70".Home_SQ;
END_REGION

REGION Network 30: Positive Flanke Automatik und Start ein
   RUNG wire#powerrail
      Contact( "AnwDB_OperatingModes_OP70".BA[0]."mode_auto+start" )
      P_Trig( "AnwDB_OperatingModes_OP70".BA[0].hm_fl_pos_mode_auto )
      Coil( "AnwDB_OperatingModes_OP70".BA[0]."fl_pos_mode_auto+start" )
   END_RUNG
   // the same network as SCL:
   #_w1 := "AnwDB_OperatingModes_OP70".BA[0]."mode_auto+start";
   #_w2 := #_w1 AND NOT "AnwDB_OperatingModes_OP70".BA[0].hm_fl_pos_mode_auto;   // rising edge
   "AnwDB_OperatingModes_OP70".BA[0].hm_fl_pos_mode_auto := #_w1;
   "AnwDB_OperatingModes_OP70".BA[0]."fl_pos_mode_auto+start" := #_w2;
END_REGION

REGION Network 31: Negative edge automatic and start on / Negative Flanke Automatik und Start ein
   RUNG wire#powerrail
      Contact( "AnwDB_OperatingModes_OP70".BA[0]."mode_auto+start" )
      N_Trig( "AnwDB_OperatingModes_OP70".BA[0].hm_fl_neg_mode_auto )
      Coil( "AnwDB_OperatingModes_OP70".BA[0]."fl_neg_mode_auto+start" )
   END_RUNG
   // the same network as SCL:
   #_w1 := "AnwDB_OperatingModes_OP70".BA[0]."mode_auto+start";
   #_w2 := NOT #_w1 AND "AnwDB_OperatingModes_OP70".BA[0].hm_fl_neg_mode_auto;   // falling edge
   "AnwDB_OperatingModes_OP70".BA[0].hm_fl_neg_mode_auto := #_w1;
   "AnwDB_OperatingModes_OP70".BA[0]."fl_neg_mode_auto+start" := #_w2;
END_REGION

REGION Network 32: Positive Flanke Grundstellung anfahren
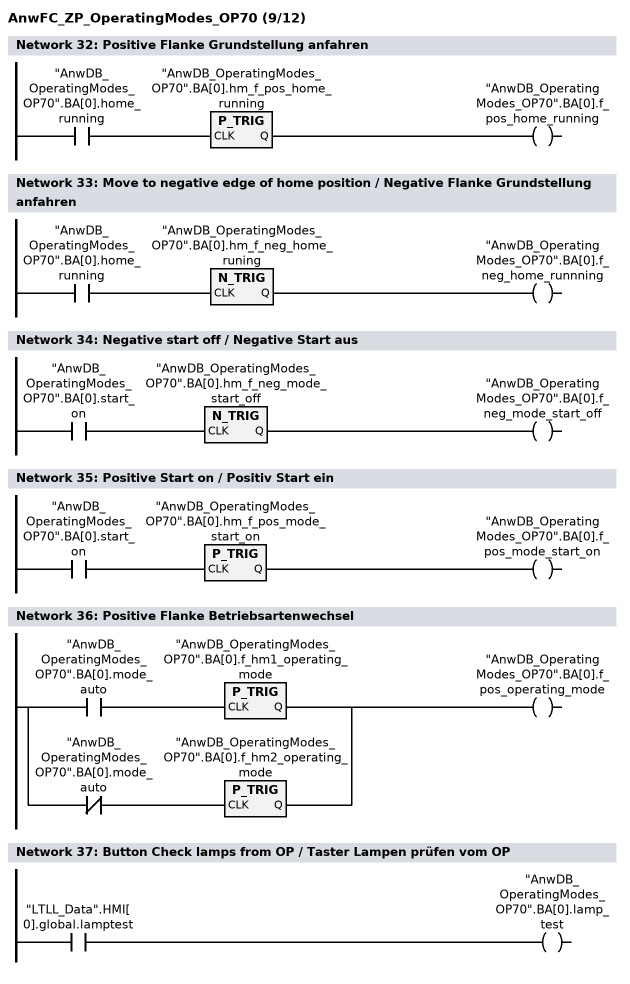
   RUNG wire#powerrail
      Contact( "AnwDB_OperatingModes_OP70".BA[0].home_running )
      P_Trig( "AnwDB_OperatingModes_OP70".BA[0].hm_f_pos_home_running )
      Coil( "AnwDB_OperatingModes_OP70".BA[0].f_pos_home_running )
   END_RUNG
   // the same network as SCL:
   #_w1 := "AnwDB_OperatingModes_OP70".BA[0].home_running;
   #_w2 := #_w1 AND NOT "AnwDB_OperatingModes_OP70".BA[0].hm_f_pos_home_running;   // rising edge
   "AnwDB_OperatingModes_OP70".BA[0].hm_f_pos_home_running := #_w1;
   "AnwDB_OperatingModes_OP70".BA[0].f_pos_home_running := #_w2;
END_REGION

REGION Network 33: Move to negative edge of home position / Negative Flanke Grundstellung anfahren
   RUNG wire#powerrail
      Contact( "AnwDB_OperatingModes_OP70".BA[0].home_running )
      N_Trig( "AnwDB_OperatingModes_OP70".BA[0].hm_f_neg_home_runing )
      Coil( "AnwDB_OperatingModes_OP70".BA[0].f_neg_home_runnning )
   END_RUNG
   // the same network as SCL:
   #_w1 := "AnwDB_OperatingModes_OP70".BA[0].home_running;
   #_w2 := NOT #_w1 AND "AnwDB_OperatingModes_OP70".BA[0].hm_f_neg_home_runing;   // falling edge
   "AnwDB_OperatingModes_OP70".BA[0].hm_f_neg_home_runing := #_w1;
   "AnwDB_OperatingModes_OP70".BA[0].f_neg_home_runnning := #_w2;
END_REGION

REGION Network 34: Negative start off / Negative Start aus
   RUNG wire#powerrail
      Contact( "AnwDB_OperatingModes_OP70".BA[0].start_on )
      N_Trig( "AnwDB_OperatingModes_OP70".BA[0].hm_f_neg_mode_start_off )
      Coil( "AnwDB_OperatingModes_OP70".BA[0].f_neg_mode_start_off )
   END_RUNG
   // the same network as SCL:
   #_w1 := "AnwDB_OperatingModes_OP70".BA[0].start_on;
   #_w2 := NOT #_w1 AND "AnwDB_OperatingModes_OP70".BA[0].hm_f_neg_mode_start_off;   // falling edge
   "AnwDB_OperatingModes_OP70".BA[0].hm_f_neg_mode_start_off := #_w1;
   "AnwDB_OperatingModes_OP70".BA[0].f_neg_mode_start_off := #_w2;
END_REGION

REGION Network 35: Positive Start on / Positiv Start ein
   RUNG wire#powerrail
      Contact( "AnwDB_OperatingModes_OP70".BA[0].start_on )
      P_Trig( "AnwDB_OperatingModes_OP70".BA[0].hm_f_pos_mode_start_on )
      Coil( "AnwDB_OperatingModes_OP70".BA[0].f_pos_mode_start_on )
   END_RUNG
   // the same network as SCL:
   #_w1 := "AnwDB_OperatingModes_OP70".BA[0].start_on;
   #_w2 := #_w1 AND NOT "AnwDB_OperatingModes_OP70".BA[0].hm_f_pos_mode_start_on;   // rising edge
   "AnwDB_OperatingModes_OP70".BA[0].hm_f_pos_mode_start_on := #_w1;
   "AnwDB_OperatingModes_OP70".BA[0].f_pos_mode_start_on := #_w2;
END_REGION

REGION Network 36: Positive Flanke Betriebsartenwechsel
   RUNG wire#powerrail
      Contact( "AnwDB_OperatingModes_OP70".BA[0].mode_auto )
      P_Trig( "AnwDB_OperatingModes_OP70".BA[0].f_hm1_operating_mode )
      wire#w1
      Coil( "AnwDB_OperatingModes_OP70".BA[0].f_pos_operating_mode )
   END_RUNG
   RUNG wire#powerrail
      I_Contact( "AnwDB_OperatingModes_OP70".BA[0].mode_auto )
      P_Trig( "AnwDB_OperatingModes_OP70".BA[0].f_hm2_operating_mode )
   END_RUNG wire#w1
   // the same network as SCL:
   #_w1 := "AnwDB_OperatingModes_OP70".BA[0].mode_auto;
   #_w2 := #_w1 AND NOT "AnwDB_OperatingModes_OP70".BA[0].f_hm1_operating_mode;   // rising edge
   "AnwDB_OperatingModes_OP70".BA[0].f_hm1_operating_mode := #_w1;
   #_w3 := NOT "AnwDB_OperatingModes_OP70".BA[0].mode_auto;
   #_w4 := #_w3 AND NOT "AnwDB_OperatingModes_OP70".BA[0].f_hm2_operating_mode;   // rising edge
   "AnwDB_OperatingModes_OP70".BA[0].f_hm2_operating_mode := #_w3;
   "AnwDB_OperatingModes_OP70".BA[0].f_pos_operating_mode := #_w2 OR #_w4;
END_REGION

REGION Network 37: Button Check lamps from OP / Taster Lampen prüfen vom OP
   RUNG wire#powerrail
      Contact( "LTLL_Data".HMI[0].global.lamptest )
      Coil( "AnwDB_OperatingModes_OP70".BA[0].lamp_test )
   END_RUNG
   // the same network as SCL:
   "AnwDB_OperatingModes_OP70".BA[0].lamp_test := "LTLL_Data".HMI[0].global.lamptest;
END_REGION

REGION Network 38: #######################MESSAGE TOUCH ####################### / ####################### MELDEANZEIGE TOUCH ######################
END_REGION

REGION Network 39: Corol Control ON HMI / Color ON HMI
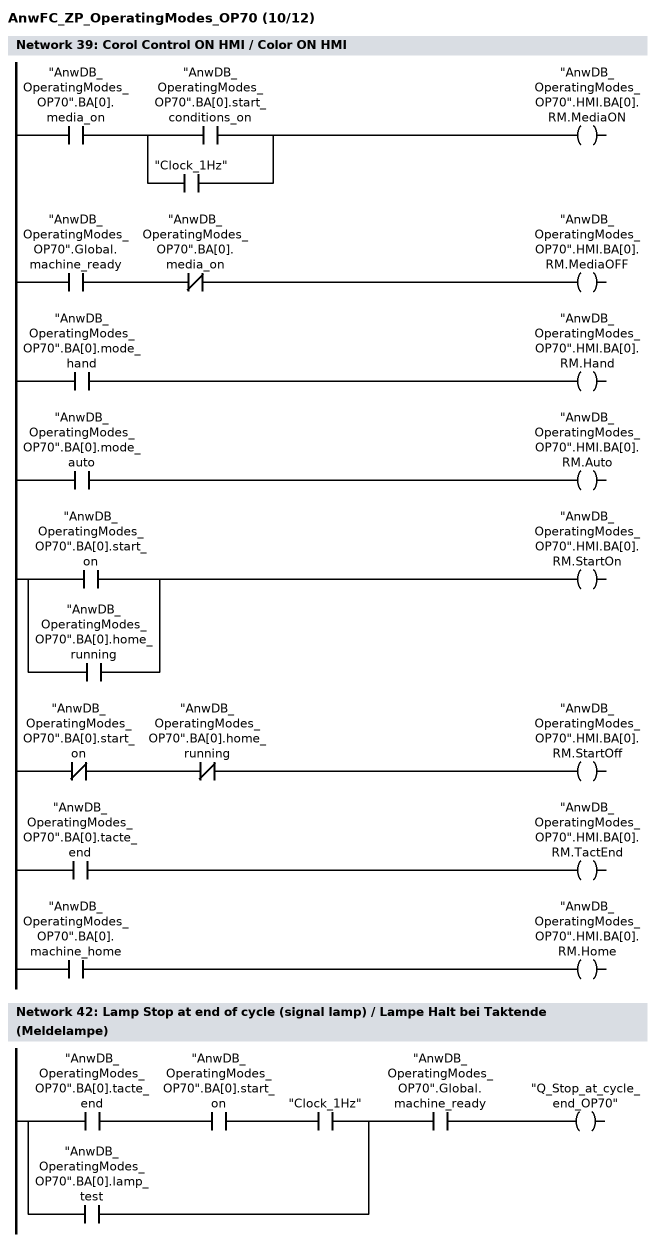
   RUNG wire#powerrail
      Contact( "AnwDB_OperatingModes_OP70".BA[0].media_on )
      wire#w1
      Contact( "AnwDB_OperatingModes_OP70".BA[0].start_conditions_on )
      wire#w2
      Coil( "AnwDB_OperatingModes_OP70".HMI.BA[0].RM.MediaON )
   END_RUNG
   RUNG wire#w1
      Contact( "Clock_1Hz" )
   END_RUNG wire#w2
   RUNG wire#powerrail
      Contact( "AnwDB_OperatingModes_OP70".Global.machine_ready )
      I_Contact( "AnwDB_OperatingModes_OP70".BA[0].media_on )
      Coil( "AnwDB_OperatingModes_OP70".HMI.BA[0].RM.MediaOFF )
   END_RUNG
   RUNG wire#powerrail
      Contact( "AnwDB_OperatingModes_OP70".BA[0].mode_hand )
      Coil( "AnwDB_OperatingModes_OP70".HMI.BA[0].RM.Hand )
   END_RUNG
   RUNG wire#powerrail
      Contact( "AnwDB_OperatingModes_OP70".BA[0].mode_auto )
      Coil( "AnwDB_OperatingModes_OP70".HMI.BA[0].RM.Auto )
   END_RUNG
   RUNG wire#powerrail
      Contact( "AnwDB_OperatingModes_OP70".BA[0].start_on )
      wire#w3
      Coil( "AnwDB_OperatingModes_OP70".HMI.BA[0].RM.StartOn )
   END_RUNG
   RUNG wire#powerrail
      Contact( "AnwDB_OperatingModes_OP70".BA[0].home_running )
   END_RUNG wire#w3
   RUNG wire#powerrail
      I_Contact( "AnwDB_OperatingModes_OP70".BA[0].start_on )
      I_Contact( "AnwDB_OperatingModes_OP70".BA[0].home_running )
      Coil( "AnwDB_OperatingModes_OP70".HMI.BA[0].RM.StartOff )
   END_RUNG
   RUNG wire#powerrail
      Contact( "AnwDB_OperatingModes_OP70".BA[0].tacte_end )
      Coil( "AnwDB_OperatingModes_OP70".HMI.BA[0].RM.TactEnd )
   END_RUNG
   RUNG wire#powerrail
      Contact( "AnwDB_OperatingModes_OP70".BA[0].machine_home )
      Coil( "AnwDB_OperatingModes_OP70".HMI.BA[0].RM.Home )
   END_RUNG
   // the same network as SCL:
   "AnwDB_OperatingModes_OP70".HMI.BA[0].RM.MediaON := "AnwDB_OperatingModes_OP70".BA[0].media_on AND ("AnwDB_OperatingModes_OP70".BA[0].start_conditions_on OR "Clock_1Hz");
   "AnwDB_OperatingModes_OP70".HMI.BA[0].RM.MediaOFF := "AnwDB_OperatingModes_OP70".Global.machine_ready AND NOT "AnwDB_OperatingModes_OP70".BA[0].media_on;
   "AnwDB_OperatingModes_OP70".HMI.BA[0].RM.Hand := "AnwDB_OperatingModes_OP70".BA[0].mode_hand;
   "AnwDB_OperatingModes_OP70".HMI.BA[0].RM.Auto := "AnwDB_OperatingModes_OP70".BA[0].mode_auto;
   "AnwDB_OperatingModes_OP70".HMI.BA[0].RM.StartOn := "AnwDB_OperatingModes_OP70".BA[0].start_on OR "AnwDB_OperatingModes_OP70".BA[0].home_running;
   "AnwDB_OperatingModes_OP70".HMI.BA[0].RM.StartOff := NOT "AnwDB_OperatingModes_OP70".BA[0].start_on AND NOT "AnwDB_OperatingModes_OP70".BA[0].home_running;
   "AnwDB_OperatingModes_OP70".HMI.BA[0].RM.TactEnd := "AnwDB_OperatingModes_OP70".BA[0].tacte_end;
   "AnwDB_OperatingModes_OP70".HMI.BA[0].RM.Home := "AnwDB_OperatingModes_OP70".BA[0].machine_home;
END_REGION

REGION Network 40: ####################### MESSAGE Pannel Button ###################### / ####################### MELDEANZEIGE ZP ######################
END_REGION

REGION Network 41: Lamp Automatic selected (signal lamp) / Lampe Vorwahl Automatik (Meldelampe)
END_REGION

REGION Network 42: Lamp Stop at end of cycle (signal lamp) / Lampe Halt bei Taktende (Meldelampe)
   RUNG wire#powerrail
      Contact( "AnwDB_OperatingModes_OP70".BA[0].tacte_end )
      Contact( "AnwDB_OperatingModes_OP70".BA[0].start_on )
      Contact( "Clock_1Hz" )
      wire#w1
      Contact( "AnwDB_OperatingModes_OP70".Global.machine_ready )
      Coil( "Q_Stop_at_cycle_end_OP70" )
   END_RUNG
   RUNG wire#powerrail
      Contact( "AnwDB_OperatingModes_OP70".BA[0].lamp_test )
   END_RUNG wire#w1
   // the same network as SCL:
   "Q_Stop_at_cycle_end_OP70" := (("AnwDB_OperatingModes_OP70".BA[0].tacte_end AND "AnwDB_OperatingModes_OP70".BA[0].start_on AND "Clock_1Hz") OR "AnwDB_OperatingModes_OP70".BA[0].lamp_test) AND "AnwDB_OperatingModes_OP70".Global.machine_ready;
END_REGION

REGION Network 43: Lamp Machine in home position (signal lamp) / Lampe Maschine in Grundstellung (Meldelampe)
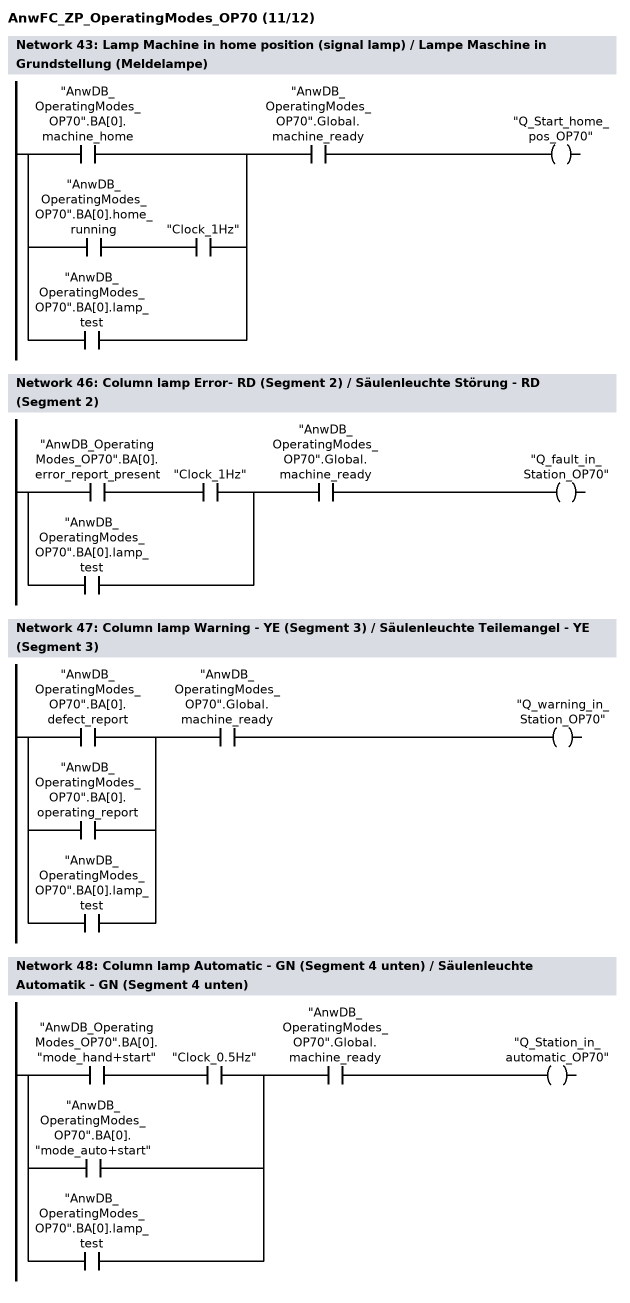
   RUNG wire#powerrail
      Contact( "AnwDB_OperatingModes_OP70".BA[0].machine_home )
      wire#w1
      Contact( "AnwDB_OperatingModes_OP70".Global.machine_ready )
      Coil( "Q_Start_home_pos_OP70" )
   END_RUNG
   RUNG wire#powerrail
      Contact( "AnwDB_OperatingModes_OP70".BA[0].home_running )
      Contact( "Clock_1Hz" )
   END_RUNG wire#w1
   RUNG wire#powerrail
      Contact( "AnwDB_OperatingModes_OP70".BA[0].lamp_test )
   END_RUNG wire#w1
   // the same network as SCL:
   "Q_Start_home_pos_OP70" := ("AnwDB_OperatingModes_OP70".BA[0].machine_home OR ("AnwDB_OperatingModes_OP70".BA[0].home_running AND "Clock_1Hz") OR "AnwDB_OperatingModes_OP70".BA[0].lamp_test) AND "AnwDB_OperatingModes_OP70".Global.machine_ready;
END_REGION

REGION Network 44: Acknowledge fault signal lamp (signal lamp) / Meldeleuchte Störung quittieren(Meldelampe)
END_REGION

REGION Network 45: ####################### SIGNAL LAMPS ###################### / ####################### MELDESÄULE ######################
END_REGION

REGION Network 46: Column lamp Error- RD (Segment 2) / Säulenleuchte Störung - RD (Segment 2)
   RUNG wire#powerrail
      Contact( "AnwDB_OperatingModes_OP70".BA[0].error_report_present )
      Contact( "Clock_1Hz" )
      wire#w1
      Contact( "AnwDB_OperatingModes_OP70".Global.machine_ready )
      Coil( "Q_fault_in_Station_OP70" )
   END_RUNG
   RUNG wire#powerrail
      Contact( "AnwDB_OperatingModes_OP70".BA[0].lamp_test )
   END_RUNG wire#w1
   // the same network as SCL:
   "Q_fault_in_Station_OP70" := (("AnwDB_OperatingModes_OP70".BA[0].error_report_present AND "Clock_1Hz") OR "AnwDB_OperatingModes_OP70".BA[0].lamp_test) AND "AnwDB_OperatingModes_OP70".Global.machine_ready;
END_REGION

REGION Network 47: Column lamp Warning - YE (Segment 3) / Säulenleuchte Teilemangel - YE (Segment 3)
   RUNG wire#powerrail
      Contact( "AnwDB_OperatingModes_OP70".BA[0].defect_report )
      wire#w1
      Contact( "AnwDB_OperatingModes_OP70".Global.machine_ready )
      Coil( "Q_warning_in_Station_OP70" )
   END_RUNG
   RUNG wire#powerrail
      Contact( "AnwDB_OperatingModes_OP70".BA[0].operating_report )
   END_RUNG wire#w1
   RUNG wire#powerrail
      Contact( "AnwDB_OperatingModes_OP70".BA[0].lamp_test )
   END_RUNG wire#w1
   // the same network as SCL:
   "Q_warning_in_Station_OP70" := ("AnwDB_OperatingModes_OP70".BA[0].defect_report OR "AnwDB_OperatingModes_OP70".BA[0].operating_report OR "AnwDB_OperatingModes_OP70".BA[0].lamp_test) AND "AnwDB_OperatingModes_OP70".Global.machine_ready;
END_REGION

REGION Network 48: Column lamp Automatic - GN (Segment 4 unten) / Säulenleuchte Automatik - GN (Segment 4 unten)
   RUNG wire#powerrail
      Contact( "AnwDB_OperatingModes_OP70".BA[0]."mode_hand+start" )
      Contact( "Clock_0.5Hz" )
      wire#w1
      Contact( "AnwDB_OperatingModes_OP70".Global.machine_ready )
      Coil( "Q_Station_in_automatic_OP70" )
   END_RUNG
   RUNG wire#powerrail
      Contact( "AnwDB_OperatingModes_OP70".BA[0]."mode_auto+start" )
   END_RUNG wire#w1
   RUNG wire#powerrail
      Contact( "AnwDB_OperatingModes_OP70".BA[0].lamp_test )
   END_RUNG wire#w1
   // the same network as SCL:
   "Q_Station_in_automatic_OP70" := (("AnwDB_OperatingModes_OP70".BA[0]."mode_hand+start" AND "Clock_0.5Hz") OR "AnwDB_OperatingModes_OP70".BA[0]."mode_auto+start" OR "AnwDB_OperatingModes_OP70".BA[0].lamp_test) AND "AnwDB_OperatingModes_OP70".Global.machine_ready;
END_REGION

REGION Network 49: ####################### Energy Counter ######################
END_REGION

REGION Network 50: Energy Counter
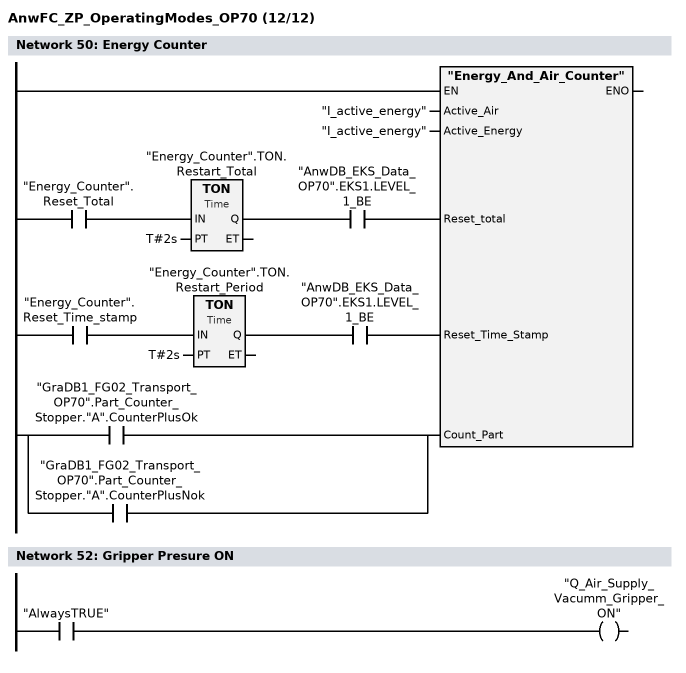
   RUNG wire#powerrail
      "Energy_And_Air_Counter"(Reset_total := wire#w1, Reset_Time_Stamp := wire#w2, Count_Part := wire#w3, Active_Air := "I_active_energy", Active_Energy := "I_active_energy")
   END_RUNG
   RUNG wire#powerrail
      Contact( "Energy_Counter".Reset_Total )
      { S7_Templates := "time_type := Time" } "Energy_Counter".TON.Restart_Total.TON(pt := T#2s, et =>)
      Contact( "AnwDB_EKS_Data_OP70".EKS1.LEVEL_1_BE )
   END_RUNG wire#w1
   RUNG wire#powerrail
      Contact( "Energy_Counter".Reset_Time_stamp )
      { S7_Templates := "time_type := Time" } "Energy_Counter".TON.Restart_Period.TON(pt := T#2s, et =>)
      Contact( "AnwDB_EKS_Data_OP70".EKS1.LEVEL_1_BE )
   END_RUNG wire#w2
   RUNG wire#powerrail
      Contact( "GraDB1_FG02_Transport_OP70".Part_Counter_Stopper."A".CounterPlusOk )
   END_RUNG wire#w3
   RUNG wire#powerrail
      Contact( "GraDB1_FG02_Transport_OP70".Part_Counter_Stopper."A".CounterPlusNok )
   END_RUNG wire#w3
   // the same network as SCL:
   "Energy_Counter".TON.Restart_Total.TON(IN := "Energy_Counter".Reset_Total, PT := T#2s);
   "Energy_Counter".TON.Restart_Period.TON(IN := "Energy_Counter".Reset_Time_stamp, PT := T#2s);
   "Energy_And_Air_Counter"(Active_Air := "I_active_energy",
                           Active_Energy := "I_active_energy",
                           Reset_total := "Energy_Counter".TON.Restart_Total.Q AND "AnwDB_EKS_Data_OP70".EKS1.LEVEL_1_BE,
                           Reset_Time_Stamp := "Energy_Counter".TON.Restart_Period.Q AND "AnwDB_EKS_Data_OP70".EKS1.LEVEL_1_BE,
                           Count_Part := "GraDB1_FG02_Transport_OP70".Part_Counter_Stopper."A".CounterPlusOk OR "GraDB1_FG02_Transport_OP70".Part_Counter_Stopper."A".CounterPlusNok);
END_REGION

REGION Network 51: ####################### Gripper Presure ON ######################
END_REGION

REGION Network 52: Gripper Presure ON
   RUNG wire#powerrail
      Contact( "AlwaysTRUE" )
      Coil( "Q_Air_Supply_Vacumm_Gripper_ON" )
   END_RUNG
   // the same network as SCL:
   "Q_Air_Supply_Vacumm_Gripper_ON" := "AlwaysTRUE";
END_REGION
END_FUNCTION
